# EPICS substitutions: iocAdminLib/archiveSrc/archive_iocAdmin.substitutions
#
# iocAdmin archive sample substitutions file
#
file archive_iocAdmin.template
{
}
